// Mitsubishi GX Works2 project: BackUP_5_12_68   PLC: FX3U/FX3UC

PROGRAM MAIN
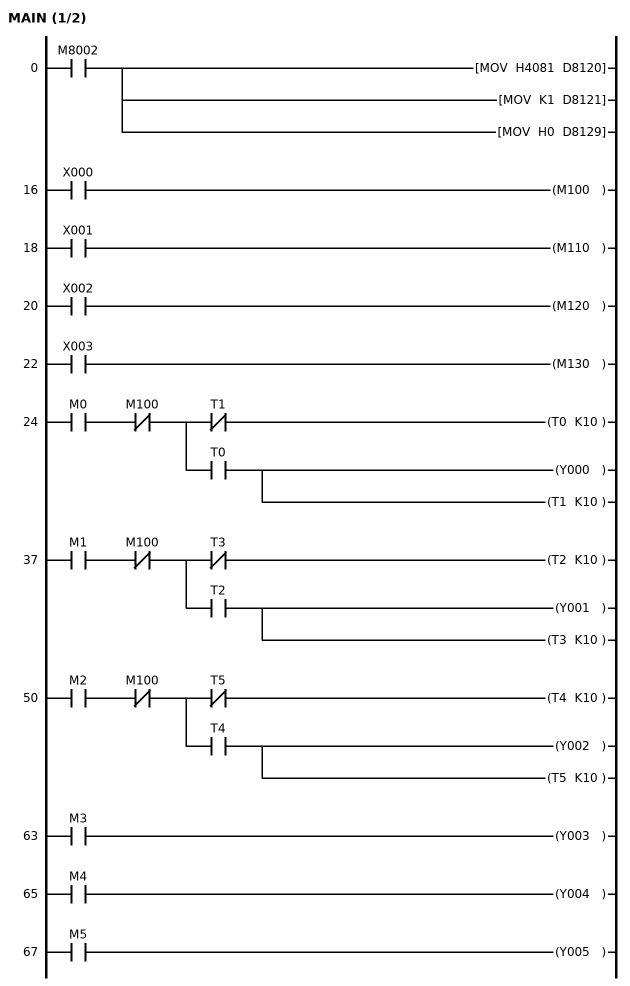
0     LD      M8002
      MOV     H4081 D8120
      MOV     K1 D8121
      MOV     H0 D8129
16    LD      X000
      OUT     M100
18    LD      X001
      OUT     M110
20    LD      X002
      OUT     M120
22    LD      X003
      OUT     M130
24    LD      M0
      ANI     M100
      MPS
      ANI     T1
      OUT     T0 K10
      MPP
      AND     T0
      OUT     Y000
      OUT     T1 K10
37    LD      M1
      ANI     M100
      MPS
      ANI     T3
      OUT     T2 K10
      MPP
      AND     T2
      OUT     Y001
      OUT     T3 K10
50    LD      M2
      ANI     M100
      MPS
      ANI     T5
      OUT     T4 K10
      MPP
      AND     T4
      OUT     Y002
      OUT     T5 K10
63    LD      M3
      OUT     Y003
65    LD      M4
      OUT     Y004
67    LD      M5
      OUT     Y005
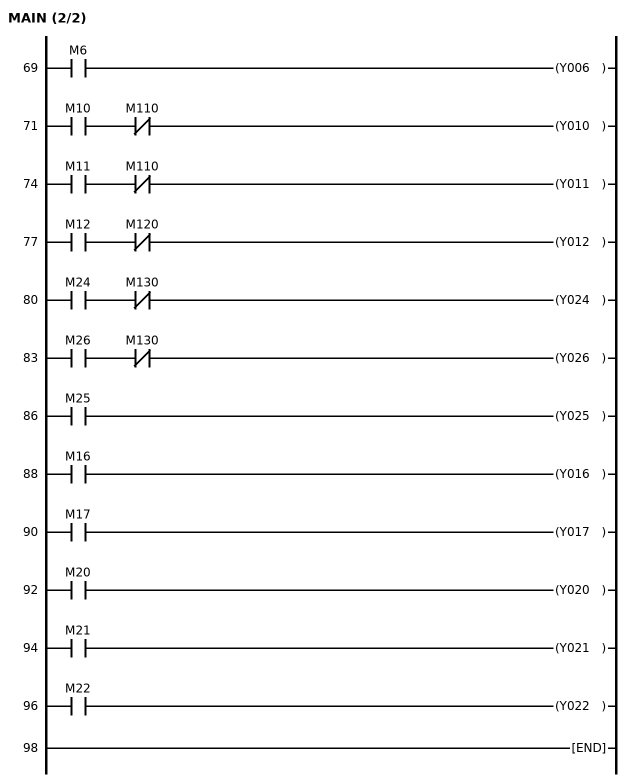
69    LD      M6
      OUT     Y006
71    LD      M10
      ANI     M110
      OUT     Y010
74    LD      M11
      ANI     M110
      OUT     Y011
77    LD      M12
      ANI     M120
      OUT     Y012
80    LD      M24
      ANI     M130
      OUT     Y024
83    LD      M26
      ANI     M130
      OUT     Y026
86    LD      M25
      OUT     Y025
88    LD      M16
      OUT     Y016
90    LD      M17
      OUT     Y017
92    LD      M20
      OUT     Y020
94    LD      M21
      OUT     Y021
96    LD      M22
      OUT     Y022
98    END
END_PROGRAM
